TYPE "CW_DIG"
VERSION : 0.1
   STRUCT
      AUTO_CMD { ExternalWritable := 'False'} : Bool;   // Auto command
      FORCE : Bool;   // Force command
      SPARE { ExternalAccessible := 'False'; ExternalVisible := 'False'; ExternalWritable := 'False'} : Bool;
      ENABLE { S7_SetPoint := 'True'} : Bool;   // Master enable
      SPARE4 { ExternalAccessible := 'False'; ExternalVisible := 'False'; ExternalWritable := 'False'} : Bool;
      INPUT { ExternalWritable := 'False'} : Bool;   // Input Status
      SPARE6 { ExternalAccessible := 'False'; ExternalVisible := 'False'; ExternalWritable := 'False'} : Bool;
      SPARE7 { ExternalAccessible := 'False'; ExternalVisible := 'False'; ExternalWritable := 'False'} : Bool;
      SPARE8 { ExternalAccessible := 'False'; ExternalVisible := 'False'; ExternalWritable := 'False'} : Bool;
      SPARE9 { ExternalAccessible := 'False'; ExternalVisible := 'False'; ExternalWritable := 'False'} : Bool;
      SPARE10 { ExternalAccessible := 'False'; ExternalVisible := 'False'; ExternalWritable := 'False'} : Bool;
      SPARE11 { ExternalAccessible := 'False'; ExternalVisible := 'False'; ExternalWritable := 'False'} : Bool;
      SPARE12 { ExternalAccessible := 'False'; ExternalVisible := 'False'; ExternalWritable := 'False'} : Bool;
      EXIST { S7_SetPoint := 'True'} : Bool;   // Exist
      OUT_ACT { ExternalWritable := 'False'} : Bool;   // Output activation
      SPARE15 { ExternalAccessible := 'False'; ExternalVisible := 'False'; ExternalWritable := 'False'} : Bool;
   END_STRUCT;

END_TYPE

TYPE "CW_MTR"
VERSION : 0.1
   STRUCT
      START_REQ { ExternalWritable := 'False'} : Bool;   // Start request
      FORCE : Bool;   // Force command
      RST_REQ : Bool;   // Reset request
      ENABLE { S7_SetPoint := 'True'} : Bool;   // Master enable
      FB_RDY { ExternalWritable := 'False'} : Bool;   // Feedback Ready/Trip
      FB_RUN { ExternalWritable := 'False'} : Bool;   // Feedback Run
      FB_RDY_EN { S7_SetPoint := 'True'} : Bool;   // Enable Ready/Trip Feedback
      FB_RUN_EN { S7_SetPoint := 'True'} : Bool;   // Enable Run Feedback
      SPARE9 { ExternalAccessible := 'False'; ExternalVisible := 'False'; ExternalWritable := 'False'} : Bool;
      NO_ERR { ExternalWritable := 'False'} : Bool;   // No error
      SRV_RST : Bool;   // Reset service interval
      SRV_IND { ExternalWritable := 'False'} : Bool;   // Service interval elapsed
      SPARE1 { ExternalAccessible := 'False'; ExternalVisible := 'False'; ExternalWritable := 'False'} : Bool;
      EXIST { S7_SetPoint := 'True'} : Bool;   // Exist
      OUT_ACT { ExternalWritable := 'False'} : Bool;   // Output activation
      SPARE2 { ExternalAccessible := 'False'; ExternalVisible := 'False'; ExternalWritable := 'False'} : Bool;
   END_STRUCT;

END_TYPE

TYPE "CW_AN"
VERSION : 0.1
   STRUCT
      SPARE0 { ExternalAccessible := 'False'; ExternalVisible := 'False'; ExternalWritable := 'False'} : Bool;
      FORCE : Bool;   // Force output
      SP_CHANGE : Bool;   // Setpoint change trigger
      ENABLE { S7_SetPoint := 'True'} : Bool;   // 1=Master enable
      SPARE4 { ExternalAccessible := 'False'; ExternalVisible := 'False'; ExternalWritable := 'False'} : Bool;
      OPEN { ExternalWritable := 'False'} : Bool;   // PLC request > 0.1
      SPARE6 { ExternalAccessible := 'False'; ExternalVisible := 'False'; ExternalWritable := 'False'} : Bool;
      SPARE7 { ExternalAccessible := 'False'; ExternalVisible := 'False'; ExternalWritable := 'False'} : Bool;
      SPARE8 { ExternalAccessible := 'False'; ExternalVisible := 'False'; ExternalWritable := 'False'} : Bool;
      NO_ERR { ExternalWritable := 'False'} : Bool;   // 1=No error
      PAR_CHANGE : Bool;   // Parameter change trigger
      SPARE11 { ExternalAccessible := 'False'; ExternalVisible := 'False'; ExternalWritable := 'False'} : Bool;
      NO { S7_SetPoint := 'True'} : Bool;   // 0=NC, 1=NO
      EXIST { S7_SetPoint := 'True'} : Bool;   // 1=Exist
      SPARE14 { ExternalAccessible := 'False'; ExternalVisible := 'False'; ExternalWritable := 'False'} : Bool;
      SPARE15 { ExternalAccessible := 'False'; ExternalVisible := 'False'; ExternalWritable := 'False'} : Bool;
   END_STRUCT;

END_TYPE

TYPE "CW_VLV"
VERSION : 0.1
   STRUCT
      AUTO_CMD { ExternalWritable := 'False'} : Bool;   // Auto command
      FORCE : Bool;   // Force command
      SPARE2 { ExternalAccessible := 'False'; ExternalVisible := 'False'; ExternalWritable := 'False'} : Bool;   // Setpoint change indication
      ENABLE { S7_SetPoint := 'True'} : Bool;   // Master enable
      FB_CLS { ExternalWritable := 'False'} : Bool;   // Feedback Close
      FB_OPN { ExternalWritable := 'False'} : Bool;   // Feedback Open
      FB_CLS_EN { S7_SetPoint := 'True'} : Bool;   // Enable Close Feedback
      FB_OPN_EN { S7_SetPoint := 'True'} : Bool;   // Enable Open Feedback
      OPN_REQ { ExternalWritable := 'False'} : Bool;   // Open Request
      NO_ERR { ExternalWritable := 'False'} : Bool;   // No error
      SRV_RST : Bool;   // Reset service interval
      SRV_IND { ExternalWritable := 'False'} : Bool;   // Service interval elapsed
      NO { S7_SetPoint := 'True'} : Bool;   // NO/NC
      EXIST { S7_SetPoint := 'True'} : Bool;   // Valve exist
      OUT_ACT { ExternalWritable := 'False'} : Bool;   // Output activation
      VLV_W_FB { S7_SetPoint := 'True'} : Bool;   // Valve without position feedbacks
   END_STRUCT;

END_TYPE

TYPE "STAT MTR"
VERSION : 0.1
   STRUCT
      TAG { ExternalWritable := 'False'; S7_SetPoint := 'True'} : String[10];   // Tag label
      CW : "CW_MTR";   // Control/Status Word
      RUN_HRS { ExternalWritable := 'False'} : UInt;   // Runtime
      FB_RUN_ADD { S7_SetPoint := 'True'} : Int := 8;   // Input address - run feedback
      FB_RDY_ADD { S7_SetPoint := 'True'} : Int := 8;   // Input address - trip feedback
      OUT_ACT_ADD { S7_SetPoint := 'True'} : Int := 8;   // Output address - activation
   END_STRUCT;

END_TYPE

TYPE "STAT VLV"
VERSION : 0.1
   STRUCT
      TAG { ExternalWritable := 'False'; S7_SetPoint := 'True'} : String[10];   // Valve tag label
      CW { S7_SetPoint := 'False'} : "CW_VLV";   // Control/Status word
      SERV_CNTR { ExternalWritable := 'False'; S7_SetPoint := 'True'} : Int;
      FB_OPN_ADD { S7_SetPoint := 'True'} : Int := 8;   // Input address - open position feedback
      FB_CLS_ADD { S7_SetPoint := 'True'} : Int := 8;   // Input address - closed position feedback
      ACT_OUT_ADD { S7_SetPoint := 'True'} : Int := 8;   // Output address - activation
   END_STRUCT;

END_TYPE

TYPE "STAT AO"
VERSION : 0.1
   STRUCT
      Tag { ExternalWritable := 'False'; S7_SetPoint := 'True'} : String[10];   // Tag label
      CW : "CW_AN";
      "Type" { ExternalAccessible := 'False'; ExternalVisible := 'False'; ExternalWritable := 'False'; S7_SetPoint := 'True'} : SInt;   // 0=V/mA, 1=Spare, 2=PN
      Address { S7_SetPoint := 'True'} : Int;   // Output Address
      Min { S7_SetPoint := 'True'} : Real;   // Scaled Min
      Max { S7_SetPoint := 'True'} : Real;   // Scaled Max
      CV : Real;   // Output value
      EU { ExternalWritable := 'False'; S7_SetPoint := 'True'} : Int;   // Eng Unit
   END_STRUCT;

END_TYPE

TYPE "STAT AI"
VERSION : 0.1
   STRUCT
      Tag { ExternalWritable := 'False'; S7_SetPoint := 'True'} : String[10];   // Tag label
      CW : "CW_AN";   // Control Word
      "Type" { S7_SetPoint := 'True'} : SInt;   // 0 = V/mA; 1 = RTD; 2=PN
      Address { S7_SetPoint := 'True'} : Int;   // Input Address
      Min { S7_SetPoint := 'True'} : Real;   // Scale min
      Max { S7_SetPoint := 'True'} : Real;   // Scale max
      PV { ExternalWritable := 'False'} : Real;   // Process value
      EU { ExternalWritable := 'False'; S7_SetPoint := 'True'} : Int;   // Engineering Units
   END_STRUCT;

END_TYPE

TYPE "STAT DI"
VERSION : 0.1
   STRUCT
      Tag { ExternalWritable := 'False'; S7_SetPoint := 'True'} : String[10];   // Tag label
      CW : "CW_DIG";
      Address { S7_SetPoint := 'True'} : Int := 8;   // Input address
   END_STRUCT;

END_TYPE

TYPE "STAT DO"
VERSION : 0.1
   STRUCT
      Tag { ExternalWritable := 'False'; S7_SetPoint := 'True'} : String[10];   // Tag label
      CW : "CW_DIG";
      Address { S7_SetPoint := 'True'} : Int := 8;   // Output address
   END_STRUCT;

END_TYPE

TYPE "STAT VFD"
VERSION : 0.1
   STRUCT
      TAG { ExternalWritable := 'False'; S7_SetPoint := 'True'} : String[10];   // Tag label
      CW : "CW_MTR";   // Control/Status Word
      "TYPE" { S7_SetPoint := 'True'} : Int;   // 0=DOL, 1=Hardwired, 2=ABB PN,  3=DANFOSS PN
      RUN_HRS { ExternalWritable := 'False'} : UInt;   // Runtime
      FB_RUN_ADD { S7_SetPoint := 'True'} : Int := 8;   // Run feedback input address
      FB_RDY_ADD { S7_SetPoint := 'True'} : Int := 8;   // Trip feedback input address
      OUT_ACT_ADD { S7_SetPoint := 'True'} : Int := 8;   // Start output address
      OUT_RST_ADD { S7_SetPoint := 'True'} : Int := 8;   // Reset output address
   END_STRUCT;

END_TYPE

TYPE "EM - 210"
VERSION : 0.1
   STRUCT
      "AV210-1" { ExternalAccessible := 'False'; ExternalVisible := 'False'; ExternalWritable := 'False'} : "STAT VLV" := ('AV210-1', ((), (), (), (), (), (), TRUE, TRUE, (), (), (), (), (), TRUE, (), TRUE), (), 184, 185, 162);   // Recirculation on/off line
      "FCV210-1" { ExternalAccessible := 'False'; ExternalVisible := 'False'; ExternalWritable := 'False'} : "STAT AO" := ('FCV210-1', ((), (), (), (), (), (), (), (), (), (), (), (), (), (), (), ()), 0, 74, (), 100.0, (), 5);   // Recirculation control valve
   END_STRUCT;

END_TYPE

TYPE "EM - 375"
VERSION : 0.1
   STRUCT
      "AV37X-1" { ExternalAccessible := 'False'; ExternalVisible := 'False'; ExternalWritable := 'False'} : "STAT VLV" := ('AV375-1', ((), (), (), TRUE, (), (), (), (), (), (), (), (), (), TRUE, (), ()), (), 8, 8, 325);   // Op. water supply
      LS793 { ExternalAccessible := 'False'; ExternalVisible := 'False'; ExternalWritable := 'False'} : "STAT DI" := ('LS793', ((), (), (), (), (), (), (), (), (), (), (), (), (), True, (), ()), 167);   // Make-up water level
      "PIS375-1" { ExternalAccessible := 'False'; ExternalVisible := 'False'; ExternalWritable := 'False'} : "STAT DI" := ('PIS375-1', ((), (), (), TRUE, (), (), (), (), (), (), (), (), (), TRUE, (), ()), 165);   // Op. water pressure
      "PT37X-1" { ExternalAccessible := 'False'; ExternalVisible := 'False'; ExternalWritable := 'False'} : "STAT AI" := ('PT376-1', ((), (), (), (), (), (), (), (), (), (), (), (), (), True, (), ()), 0, 102, 0.0, 1000.0, (), ());   // Op. water pressure
   END_STRUCT;

END_TYPE

TYPE "EM - 506"
VERSION : 0.1
   STRUCT
      "AV543-1" { ExternalAccessible := 'False'; ExternalVisible := 'False'; ExternalWritable := 'False'} : "STAT VLV" := ('AV543-1', ((), (), (), (), (), (), TRUE, TRUE, (), (), (), (), TRUE, TRUE, (), TRUE), (), 220, 221, 180);   // Cyclone vent pipe
      IP506a { ExternalAccessible := 'False'; ExternalVisible := 'False'; ExternalWritable := 'False'} : "STAT AO" := ('IP506A', ((), (), (), (), (), (), (), (), (), (), (), (), (), True, (), ()), (), 68, (), 100.0, (), 5);   // Discharge pressure
      "PV376-1" { ExternalAccessible := 'False'; ExternalVisible := 'False'; ExternalWritable := 'False'} : "STAT VLV" := ('PV376-1', ((), (), (), (), (), (), (), (), (), (), (), (), (), TRUE, (), ()), (), 8, 8, 337);   // Op. water supply
      "PV376-2" { ExternalAccessible := 'False'; ExternalVisible := 'False'; ExternalWritable := 'False'} : "STAT VLV" := ('PV376-2', ((), (), (), (), (), (), (), (), (), (), (), (), (), TRUE, (), ()), (), 8, 8, 340);   // Op. water supply
      AVDCH { ExternalAccessible := 'False'; ExternalVisible := 'False'; ExternalWritable := 'False'} : "STAT VLV" := ('506c', ((), (), (), TRUE, (), (), (), (), (), (), (), (), (), TRUE, (), ()), (), (), (), 332);   // Large discharge
   END_STRUCT;

END_TYPE

TYPE "EM - P201"
VERSION : 0.1
   STRUCT
      "P201-1" { ExternalAccessible := 'False'; ExternalVisible := 'False'; ExternalWritable := 'False'} : "STAT VFD" := ('P201-1', ((), (), (), (), (), (), TRUE, TRUE, (), (), (), (), (), TRUE, (), ()), 1, (), 346, 347, 246, 247);   // Feed pump
      "P201-1_SPEED_REF" { ExternalAccessible := 'False'; ExternalVisible := 'False'; ExternalWritable := 'False'} : "STAT AO" := ((), ((), (), (), (), (), (), (), (), (), (), (), (), (), (), (), ()), (), 82, (), 100.0, (), 5);
      "TS201-1" { ExternalAccessible := 'False'; ExternalVisible := 'False'; ExternalWritable := 'False'} : "STAT DI" := ('TS201-1', ((), (), (), (), (), (), (), (), (), (), (), (), (), (), (), ()), ());   // PTC for feed pump motor
   END_STRUCT;

END_TYPE

TYPE "EM - 208"
VERSION : 0.1
   STRUCT
      "AV208-1" { ExternalAccessible := 'False'; ExternalVisible := 'False'; ExternalWritable := 'False'} : "STAT VLV" := ('AV208-1', ((), (), (), (), (), (), TRUE, TRUE, (), (), (), (), (), (), (), TRUE), (), 182, 183, 161);   // Blending line on/off valve
      "FCV208-1" { ExternalAccessible := 'False'; ExternalVisible := 'False'; ExternalWritable := 'False'} : "STAT AO" := ('FCV208-1', ((), (), (), (), (), (), (), (), (), (), (), (), (), (), (), ()), 0, 72, (), 100.0, (), 5);   // Blending flow control valve
      "FIT208-1" { ExternalAccessible := 'False'; ExternalVisible := 'False'; ExternalWritable := 'False'} : "STAT AI" := ('FIT208-1', ((), (), (), (), (), (), (), (), (), (), (), (), (), (), (), ()), (), (), (), (), (), ());   // Blending flow meter
      "P208-1" { ExternalAccessible := 'False'; ExternalVisible := 'False'; ExternalWritable := 'False'} : "STAT MTR" := ('P208-1', ((), (), (), (), (), (), TRUE, TRUE, (), (), (), (), (), TRUE, (), ()), (), 350, 351, 250);   // Blending pump
      "QT220-2" { ExternalAccessible := 'False'; ExternalVisible := 'False'; ExternalWritable := 'False'} : "STAT AI" := ('QT220-2', ((), (), (), (), (), (), (), (), (), (), (), (), (), (), (), ()), 0, 86, 0.0, 1000.0, (), ());   // Blending turbidity
      "QT220-2_OK" { ExternalAccessible := 'False'; ExternalVisible := 'False'; ExternalWritable := 'False'} : "STAT DI" := ((), ((), (), (), (), (), (), (), (), (), (), (), (), (), (), (), ()), 173);   // Turbicity sensor status
   END_STRUCT;

END_TYPE

TYPE "EM - 300"
VERSION : 0.1
   STRUCT
      "AV301-1" { ExternalAccessible := 'False'; ExternalVisible := 'False'; ExternalWritable := 'False'} : "STAT VLV" := ('AV301-1', ((), (), (), TRUE, (), (), TRUE, TRUE, (), (), (), (), (), TRUE, (), TRUE), (), 200, 201, 170);   // Flush water supply
      "AV302a-1" { ExternalAccessible := 'False'; ExternalVisible := 'False'; ExternalWritable := 'False'} : "STAT VLV" := ('AV302a-1', ((), (), (), (), (), (), (), (), (), (), (), (), (), (), (), ()), (), (), (), 164);   // Flush above bowl
      "AV302-1" { ExternalAccessible := 'False'; ExternalVisible := 'False'; ExternalWritable := 'False'} : "STAT VLV" := ('AV302-1', ((), (), (), (), (), (), (), (), (), (), (), (), (), TRUE, (), ()), (), 8, 8, 320);   // Flush bowl upper
      "AV303-1" { ExternalAccessible := 'False'; ExternalVisible := 'False'; ExternalWritable := 'False'} : "STAT VLV" := ('AV303-1', ((), (), (), (), (), (), (), (), (), (), (), (), (), TRUE, (), ()), (), 8, 8, 321);   // Flush bowl lower
      "AV304-1" { ExternalAccessible := 'False'; ExternalVisible := 'False'; ExternalWritable := 'False'} : "STAT VLV" := ('AV304-1', ((), (), (), (), (), (), (), (), (), (), (), (), (), TRUE, (), ()), (), 8, 8, 322);   // Flush sediment outlet
      "AV305-1" { ExternalAccessible := 'False'; ExternalVisible := 'False'; ExternalWritable := 'False'} : "STAT VLV" := ('AV305-1', ((), (), (), (), (), (), (), (), (), (), (), (), (), TRUE, (), ()), (), 8, 8, 323);   // Flush cyclone
      "AV306-1" { ExternalAccessible := 'False'; ExternalVisible := 'False'; ExternalWritable := 'False'} : "STAT VLV" := ('AV306-1', ((), (), (), (), (), (), (), (), (), (), (), (), (), TRUE, (), ()), (), 8, 8, 324);   // Flush cyclone vent pipe
      "AV320-1" { ExternalAccessible := 'False'; ExternalVisible := 'False'; ExternalWritable := 'False'} : "STAT VLV" := ('AV320-1', ((), (), (), (), (), (), TRUE, TRUE, (), (), (), (), (), TRUE, (), TRUE), (), 202, 203, 171);   // CIP flush supply
      "AV635-1" { ExternalAccessible := 'False'; ExternalVisible := 'False'; ExternalWritable := 'False'} : "STAT VLV" := ('AV635-1', ((), (), (), (), (), (), (), (), (), (), (), (), (), TRUE, (), ()), (), 8, 8, 330);   // Flush outlet mechanical seals
      "PS301-1" { ExternalAccessible := 'False'; ExternalVisible := 'False'; ExternalWritable := 'False'} : "STAT DI" := ('PS301-1', ((), (), (), (), (), (), (), (), (), (), (), (), (), True, (), ()), 164);   // Water supply pressure
   END_STRUCT;

END_TYPE

TYPE "EM - PRU2"
VERSION : 0.1
   STRUCT
      "AV460b-1" { ExternalAccessible := 'False'; ExternalVisible := 'False'; ExternalWritable := 'False'} : "STAT VLV" := ('AV460b-1', ((), (), (), (), (), (), (), (), (), (), (), (), TRUE, TRUE, (), ()), (), (), (), 162);   // PRU tank drain
      "AV660b-1" { ExternalAccessible := 'False'; ExternalVisible := 'False'; ExternalWritable := 'False'} : "STAT VLV" := ('AV660b-1', ((), (), (), (), (), (), (), (), (), (), (), (), (), TRUE, (), ()), (), (), (), 192);   // Sealing liquid SRU pump
      "GS220-1" { ExternalAccessible := 'False'; ExternalVisible := 'False'; ExternalWritable := 'False'} : "STAT DI" := ('GS220-1', ((), (), (), (), (), (), (), (), (), (), (), (), (), (), (), ()), 186);   // PRU tank cover switch
      "FS661b-1" { ExternalAccessible := 'False'; ExternalVisible := 'False'; ExternalWritable := 'False'} : "STAT DI" := ((), ((), (), (), (), (), (), (), (), (), (), (), (), (), (), (), ()), 172);   // PRU sealing l
      "P220-1" { ExternalAccessible := 'False'; ExternalVisible := 'False'; ExternalWritable := 'False'} : "STAT VFD" := ('P220-1', ((), (), (), (), (), (), TRUE, TRUE, (), (), (), (), (), TRUE, (), ()), 2, (), (), (), 540, ());   // PRU pump
   END_STRUCT;

END_TYPE

TYPE "EM - 463"
VERSION : 0.1
   STRUCT
      "AV305-2" { ExternalAccessible := 'False'; ExternalVisible := 'False'; ExternalWritable := 'False'} : "STAT VLV" := ('AV305-2', ((), (), (), (), (), (), (), (), (), (), (), (), (), TRUE, (), ()), (), 8, 8, 345);   // Tank flush - CIP
      "AV463-1" { ExternalAccessible := 'False'; ExternalVisible := 'False'; ExternalWritable := 'False'} : "STAT VLV" := ('AV463-1', ((), (), (), (), (), (), TRUE, TRUE, (), (), (), (), TRUE, TRUE, (), TRUE), (), 224, 225, 182);   // Inlet valve
      "AV463-2" { ExternalAccessible := 'False'; ExternalVisible := 'False'; ExternalWritable := 'False'} : "STAT VLV" := ('AV463-2', ((), (), (), (), (), (), TRUE, TRUE, (), (), (), (), (), TRUE, (), TRUE), (), 226, 227, 183);   // Overflow outlet valve
      "AV470-1" { ExternalAccessible := 'False'; ExternalVisible := 'False'; ExternalWritable := 'False'} : "STAT VLV" := ('AV470-1', ((), (), (), (), (), (), (), (), (), (), (), (), TRUE, TRUE, (), ()), (), 8, 8, 342);   // Pressure relief valve
      "AV660-1" { ExternalAccessible := 'False'; ExternalVisible := 'False'; ExternalWritable := 'False'} : "STAT VLV" := ('AV660-1', ((), (), (), (), (), (), (), (), (), (), (), (), (), TRUE, (), ()), (), 8, 8, 341);   // Vacuum pump sealing water
      "AV660-2" { ExternalAccessible := 'False'; ExternalVisible := 'False'; ExternalWritable := 'False'} : "STAT VLV" := ('AV660-2', ((), (), (), (), (), (), (), (), (), (), (), (), (), TRUE, (), ()), (), 8, 8, 346);   // Tank flush - water
      "LT463-1" { ExternalAccessible := 'False'; ExternalVisible := 'False'; ExternalWritable := 'False'} : "STAT AI" := ('LT463-1', ((), (), (), (), (), (), (), (), (), (), (), (), (), (), (), ()), (), 82, (), 100.0, (), ());   // Tank level
      "PIT463-1" { ExternalAccessible := 'False'; ExternalVisible := 'False'; ExternalWritable := 'False'} : "STAT AI" := ('PIT463-1', ((), (), (), (), (), (), (), (), (), (), (), (), (), (), (), ()), (), 84, -100.0, 1000.0, (), ());   // eMotion pressure
      "P463-1" { ExternalAccessible := 'False'; ExternalVisible := 'False'; ExternalWritable := 'False'} : "STAT MTR" := ('P463-1', ((), (), (), (), (), (), TRUE, TRUE, (), (), (), (), (), TRUE, (), ()), (), 344, 345, 245);   // Vacuum pump
   END_STRUCT;

END_TYPE

TYPE "EM - 551"
VERSION : 0.1
   STRUCT
      "FIT551-1" { ExternalAccessible := 'False'; ExternalVisible := 'False'; ExternalWritable := 'False'} : "STAT AI" := ('FIT551-1', ((), (), (), (), (), (), (), (), (), (), (), (), (), (), (), ()), (), 66, (), 70700.0, (), ());   // ProCarb CO2 flowmeter
      "FCV551-1" { ExternalAccessible := 'False'; ExternalVisible := 'False'; ExternalWritable := 'False'} : "STAT AO" := ('FCV551-1', ((), (), (), (), (), (), (), (), (), (), (), (), (), (), (), ()), (), 66, (), 100.0, (), 5);   // ProCarb CO2 flow control valve
   END_STRUCT;

END_TYPE

TYPE "EM - PRU1"
VERSION : 0.1
   STRUCT
      "AV461b-1" { ExternalAccessible := 'False'; ExternalVisible := 'False'; ExternalWritable := 'False'} : "STAT VLV" := ('AV461b-1', ((), (), (), (), (), (), (), (), (), (), (), (), TRUE, TRUE, (), ()), (), (), (), 163);   // PRU tank drain
      "AV660a-1" { ExternalAccessible := 'False'; ExternalVisible := 'False'; ExternalWritable := 'False'} : "STAT VLV" := ('AV660a-1', ((), (), (), (), (), (), (), (), (), (), (), (), (), TRUE, (), ()), (), (), (), 191);   // Sealing liquid SRU pump
      "GS221-1" { ExternalAccessible := 'False'; ExternalVisible := 'False'; ExternalWritable := 'False'} : "STAT DI" := ('GS221-1', ((), (), (), (), (), (), (), (), (), (), (), (), (), (), (), ()), 187);   // PRU cover switch
      "FS661a-1" { ExternalAccessible := 'False'; ExternalVisible := 'False'; ExternalWritable := 'False'} : "STAT DI" := ((), ((), (), (), (), (), (), (), (), (), (), (), (), (), (), (), ()), 171);
      "P221-1" { ExternalAccessible := 'False'; ExternalVisible := 'False'; ExternalWritable := 'False'} : "STAT VFD" := ('P221-1', ((), (), (), (), (), (), TRUE, TRUE, (), (), (), (), (), TRUE, (), ()), 2, (), (), (), 532, ());   // PRU pump
   END_STRUCT;

END_TYPE

TYPE "EM - 222"
VERSION : 0.1
   STRUCT
      "AV222-1" { ExternalAccessible := 'False'; ExternalVisible := 'False'; ExternalWritable := 'False'} : "STAT VLV" := ('AV222-1', ((), (), (), (), (), (), TRUE, TRUE, (), (), (), (), (), TRUE, (), TRUE), (), 194, 195, 166);   // Soilds outlet change-over valve
      "LS222-1" { ExternalAccessible := 'False'; ExternalVisible := 'False'; ExternalWritable := 'False'} : "STAT DI" := ('LS222-1', ((), (), (), TRUE, (), (), (), (), (), (), (), (), (), True, (), ()), 326);   // Level in cyclone high-high
      "LS222-2" { ExternalAccessible := 'False'; ExternalVisible := 'False'; ExternalWritable := 'False'} : "STAT DI" := ('LS222-2', ((), (), (), (), (), (), (), (), (), (), (), (), (), (), (), ()), 327);   // Level in cylone high
      "LS222-3" { ExternalAccessible := 'False'; ExternalVisible := 'False'; ExternalWritable := 'False'} : "STAT DI" := ('LS222-3', ((), (), (), (), (), (), (), (), (), (), (), (), (), (), (), ()), 330);   // Level in cyclone low
      "P222-1" { ExternalAccessible := 'False'; ExternalVisible := 'False'; ExternalWritable := 'False'} : "STAT MTR" := ('P222-1', ((), (), (), TRUE, (), (), TRUE, TRUE, (), (), (), (), (), True, (), ()), (), 334, 335, 242);   // Solids pump
      "PIT222-1" { ExternalAccessible := 'False'; ExternalVisible := 'False'; ExternalWritable := 'False'} : "STAT AI" := ('PIT222-1', ((), (), (), (), (), (), (), (), (), (), (), (), (), (), (), ()), (), 78, (), 1000.0, (), ());   // Solids pressure
      "TS222-1" { ExternalAccessible := 'False'; ExternalVisible := 'False'; ExternalWritable := 'False'} : "STAT DI" := ('TS222-1', ((), (), (), TRUE, (), (), (), (), (), (), (), (), (), TRUE, (), ()), 324);   // Solids pump dry-run potection
      "TT222-1" { ExternalAccessible := 'False'; ExternalVisible := 'False'; ExternalWritable := 'False'} : "STAT AI" := ('TT222-1', ((), (), (), (), (), (), (), (), (), (), (), (), (), (), (), ()), 1, 134, 0.0, 200.0, (), ());   // Solids pump stator temperature
   END_STRUCT;

END_TYPE

TYPE "EM - BC-COMM"
VERSION : 0.1
   STRUCT
      BCI0 { ExternalAccessible := 'False'; ExternalVisible := 'False'; ExternalWritable := 'False'; S7_SetPoint := 'True'} : Int := 173;   // BC I/O CMD
      BCI1 { ExternalAccessible := 'False'; ExternalVisible := 'False'; ExternalWritable := 'False'; S7_SetPoint := 'True'} : Int := 174;   // BC I/O CMD
      BCI2 { ExternalAccessible := 'False'; ExternalVisible := 'False'; ExternalWritable := 'False'; S7_SetPoint := 'True'} : Int := 175;   // BC I/O CMD
      BCI3 { ExternalAccessible := 'False'; ExternalVisible := 'False'; ExternalWritable := 'False'; S7_SetPoint := 'True'} : Int := 176;   // BC I/O CMD
      BCO0 { ExternalAccessible := 'False'; ExternalVisible := 'False'; ExternalWritable := 'False'; S7_SetPoint := 'True'} : Int := 185;   // BC I/O STATUS
      BCO1 { ExternalAccessible := 'False'; ExternalVisible := 'False'; ExternalWritable := 'False'; S7_SetPoint := 'True'} : Int := 186;   // BC I/O STATUS
      BCO2 { ExternalAccessible := 'False'; ExternalVisible := 'False'; ExternalWritable := 'False'; S7_SetPoint := 'True'} : Int := 187;   // BC I/O STATUS
      BCO3 { ExternalAccessible := 'False'; ExternalVisible := 'False'; ExternalWritable := 'False'; S7_SetPoint := 'True'} : Int := 190;   // BC I/O STATUS
      ALARM { ExternalAccessible := 'False'; ExternalVisible := 'False'; ExternalWritable := 'False'; S7_SetPoint := 'True'} : Int := 197;   // BC I/O STATUS
   END_STRUCT;

END_TYPE

TYPE "EM - RCB"
VERSION : 0.1
   STRUCT
      "RCB_IN_Dch 1" { ExternalAccessible := 'False'; ExternalVisible := 'False'; ExternalWritable := 'False'; S7_SetPoint := 'True'} : Int := 200;   // RCB CMD
      "RCB_IN_Dch 2" { ExternalAccessible := 'False'; ExternalVisible := 'False'; ExternalWritable := 'False'; S7_SetPoint := 'True'} : Int := 201;   // RCB CMD
      RCB_IN_ZoomIn { ExternalAccessible := 'False'; ExternalVisible := 'False'; ExternalWritable := 'False'; S7_SetPoint := 'True'} : Int := 202;   // RCB CMD
      RCB_IN_Prod { ExternalAccessible := 'False'; ExternalVisible := 'False'; ExternalWritable := 'False'; S7_SetPoint := 'True'} : Int := 203;   // RCB CMD
      RCB_IN_WaterTest { ExternalAccessible := 'False'; ExternalVisible := 'False'; ExternalWritable := 'False'; S7_SetPoint := 'True'} : Int := 204;   // RCB CMD
      RCB_IN_CipWater { ExternalAccessible := 'False'; ExternalVisible := 'False'; ExternalWritable := 'False'; S7_SetPoint := 'True'} : Int := 205;   // RCB CMD
      RCB_IN_ZoomOut { ExternalAccessible := 'False'; ExternalVisible := 'False'; ExternalWritable := 'False'; S7_SetPoint := 'True'} : Int := 206;   // RCB CMD
      RCB_IN_Start { ExternalAccessible := 'False'; ExternalVisible := 'False'; ExternalWritable := 'False'; S7_SetPoint := 'True'} : Int := 207;   // RCB CMD
      RCB_IN_Stop { ExternalAccessible := 'False'; ExternalVisible := 'False'; ExternalWritable := 'False'; S7_SetPoint := 'True'} : Int := 210;   // RCB CMD
      ExtInterlockStart { ExternalAccessible := 'False'; ExternalVisible := 'False'; ExternalWritable := 'False'; S7_SetPoint := 'True'} : Int := 160;   // INTERLOCKS
      ExtInterlockProd { ExternalAccessible := 'False'; ExternalVisible := 'False'; ExternalWritable := 'False'; S7_SetPoint := 'True'} : Int := 161;   // INTERLOCKS
      ExtInterlockCIP { ExternalAccessible := 'False'; ExternalVisible := 'False'; ExternalWritable := 'False'; S7_SetPoint := 'True'} : Int := 162;   // INTERLOCKS
      "RCB_OUT_Dch 1" { ExternalAccessible := 'False'; ExternalVisible := 'False'; ExternalWritable := 'False'; S7_SetPoint := 'True'} : Int := 160;   // RCB STATUS
      "RCB_OUT_Dch 2" { ExternalAccessible := 'False'; ExternalVisible := 'False'; ExternalWritable := 'False'; S7_SetPoint := 'True'} : Int := 161;   // RCB STATUS
      RCB_OUT_ZoomIn { ExternalAccessible := 'False'; ExternalVisible := 'False'; ExternalWritable := 'False'; S7_SetPoint := 'True'} : Int := 162;   // RCB STATUS
      RCB_OUT_Prod { ExternalAccessible := 'False'; ExternalVisible := 'False'; ExternalWritable := 'False'; S7_SetPoint := 'True'} : Int := 163;   // RCB STATUS
      RCB_OUT_WaterTest { ExternalAccessible := 'False'; ExternalVisible := 'False'; ExternalWritable := 'False'; S7_SetPoint := 'True'} : Int := 164;   // RCB STATUS
      RCB_OUT_CipWater { ExternalAccessible := 'False'; ExternalVisible := 'False'; ExternalWritable := 'False'; S7_SetPoint := 'True'} : Int := 165;   // RCB STATUS
      RCB_OUT_ZoomOut { ExternalAccessible := 'False'; ExternalVisible := 'False'; ExternalWritable := 'False'; S7_SetPoint := 'True'} : Int := 166;   // RCB STATUS
      RCB_OUT_Start { ExternalAccessible := 'False'; ExternalVisible := 'False'; ExternalWritable := 'False'; S7_SetPoint := 'True'} : Int := 167;   // RCB STATUS
      RCB_OUT_Stop { ExternalAccessible := 'False'; ExternalVisible := 'False'; ExternalWritable := 'False'; S7_SetPoint := 'True'} : Int := 170;   // RCB STATUS
   END_STRUCT;

END_TYPE

TYPE "EM - 430"
VERSION : 0.1
   STRUCT
      "AV400-1" { ExternalAccessible := 'False'; ExternalVisible := 'False'; ExternalWritable := 'False'} : "STAT VLV" := ('AV400-1', ((), (), (), (), (), (), (), (), (), (), (), (), (), TRUE, (), ()), (), 8, 8, 8);   // Cooling liquid supply
      "AV430-1" { ExternalAccessible := 'False'; ExternalVisible := 'False'; ExternalWritable := 'False'} : "STAT VLV" := ('AV430-1', ((), (), (), (), (), (), (), (), (), (), (), (), (), TRUE, (), ()), (), 8, 8, 343);   // Glycol supply
      "FCV430-1" { ExternalAccessible := 'False'; ExternalVisible := 'False'; ExternalWritable := 'False'} : "STAT AO" := ('FCV430-1', ((), (), (), (), (), (), (), (), (), (), (), (), (), (), (), ()), (), 76, (), 100.0, (), 5);   // Glycol flow control valve
      "LT406-1" { ExternalAccessible := 'False'; ExternalVisible := 'False'; ExternalWritable := 'False'} : "STAT AI" := ('LT406-1', ((), (), (), (), (), (), (), (), (), (), (), (), (), (), (), ()), (), (), (), 100.0, (), ());   // Cooling liquid level
      "P406-1" { ExternalAccessible := 'False'; ExternalVisible := 'False'; ExternalWritable := 'False'} : "STAT MTR" := ('P406-1', ((), (), (), (), (), (), TRUE, TRUE, (), (), (), (), (), TRUE, (), ()), (), 342, 343, 244);   // Cooling liquid pump
      "TT406-1" { ExternalAccessible := 'False'; ExternalVisible := 'False'; ExternalWritable := 'False'} : "STAT AI" := ('TT406-1', ((), (), (), (), (), (), (), (), (), (), (), (), (), (), (), ()), (), 86, (), 200.0, (), ());   // Cooling liquid temperature
   END_STRUCT;

END_TYPE

TYPE "EM - 212"
VERSION : 0.1
   STRUCT
      "AV212-1" { ExternalAccessible := 'False'; ExternalVisible := 'False'; ExternalWritable := 'False'} : "STAT VLV" := ('AV212-1', ((), (), (), (), (), (), TRUE, TRUE, (), (), (), (), TRUE, TRUE, (), TRUE), (), 186, 187, 163);   // By-pass valve
   END_STRUCT;

END_TYPE

TYPE "EM - 206"
VERSION : 0.1
   STRUCT
      "AV206-1" : "STAT VLV" := ('AV206-1', ((), (), (), (), (), (), (), (), (), (), (), (), (), True, (), ()), (), 8, 8, 161);   // Brine/Centrate on/off valve
      "PIT206-1" : "STAT AI" := ('PIT206-1', ((), (), (), (), (), (), (), (), (), (), (), (), (), True, (), ()), 0, 86, 0.0, 1000.0, (), ());   // Brine/Centrate pressure
   END_STRUCT;

END_TYPE

TYPE "EM - 22X"
VERSION : 0.1
   STRUCT
      "AV220-1" { ExternalAccessible := 'False'; ExternalVisible := 'False'; ExternalWritable := 'False'} : "STAT VLV" := ('AV220-1', ((), (), (), (), (), (), TRUE, TRUE, (), (), (), (), (), TRUE, (), TRUE), (), 190, 191, 164);   // LP outlet valve
      "AV460-1" { ExternalAccessible := 'False'; ExternalVisible := 'False'; ExternalWritable := 'False'} : "STAT VLV" := ('AV460-1', ((), (), (), (), (), (), TRUE, TRUE, (), (), (), (), TRUE, TRUE, (), TRUE), (), 210, 211, 174);   // LP outlet to drain valve
      "SV220-1" { ExternalAccessible := 'False'; ExternalVisible := 'False'; ExternalWritable := 'False'} : "STAT VLV" := ('SV220-1', ((), (), (), (), (), (), (), (), (), (), (), (), (), (), (), ()), (), (), (), 333);   // Back pressure air supply
      "FIT22X-1" { ExternalAccessible := 'False'; ExternalVisible := 'False'; ExternalWritable := 'False'} : "STAT AI" := ('FIT220-1', ((), (), (), True, (), (), (), (), (), (), (), (), (), (), (), ()), (), (), (), (), (), ());   // LP outlet flowmeter
      "PIT22X-1" { ExternalAccessible := 'False'; ExternalVisible := 'False'; ExternalWritable := 'False'} : "STAT AI" := ('PIT220-1', ((), (), (), True, (), (), (), (), (), (), (), (), (), True, (), ()), 0, 66, 0.0, 1000.0, (), ());   // LP outlet pressure
      "QT220-1" { ExternalAccessible := 'False'; ExternalVisible := 'False'; ExternalWritable := 'False'} : "STAT AI" := ('QT220-1', ((), (), (), (), (), (), (), (), (), (), (), (), (), True, (), ()), 0, 70, 0.0, 100.0, (), ());   // LP outlet turbidity
      "PCV22X-1" { ExternalAccessible := 'False'; ExternalVisible := 'False'; ExternalWritable := 'False'} : "STAT AO" := ('PCV220-1', ((), (), (), True, (), (), (), (), (), (), (), (), (), True, (), ()), 0, 66, (), 100.0, (), 5);   // LP outlet pressure control valve
      "QT220-1_OK" { ExternalAccessible := 'False'; ExternalVisible := 'False'; ExternalWritable := 'False'} : "STAT DI" := ('QT220-1 OK', ((), (), (), (), (), (), (), (), (), (), (), (), (), True, (), ()), 172);   // Turbidity sensor status
      "LA220-1" { ExternalAccessible := 'False'; ExternalVisible := 'False'; ExternalWritable := 'False'} : "STAT DO" := ('LA220-1', ((), (), (), (), (), (), (), (), (), (), (), (), (), True, (), ()), 192);   // LP outlet sight glass backlight
   END_STRUCT;

END_TYPE

TYPE "EM - 100"
VERSION : 0.1
   STRUCT
      "L-GREEN" { ExternalAccessible := 'False'; ExternalVisible := 'False'; ExternalWritable := 'False'} : "STAT DO" := ('L-GREEN', ((), (), (), (), (), (), (), (), (), (), (), (), (), True, (), ()), 193);   // Green light
      "L-YELLOW" { ExternalAccessible := 'False'; ExternalVisible := 'False'; ExternalWritable := 'False'} : "STAT DO" := ('L-YELLOW', ((), (), (), (), (), (), (), (), (), (), (), (), (), True, (), ()), 194);   // Yellow light
      "L-RED" { ExternalAccessible := 'False'; ExternalVisible := 'False'; ExternalWritable := 'False'} : "STAT DO" := ('L-RED', ((), (), (), TRUE, (), (), (), (), (), (), (), (), (), TRUE, (), ()), 195);   // Red light
      "L-BUZZ" { ExternalAccessible := 'False'; ExternalVisible := 'False'; ExternalWritable := 'False'} : "STAT DO" := ('L-BUZZ', ((), (), (), TRUE, (), (), (), (), (), (), (), (), (), TRUE, (), ()), 196);   // Buzzier
      EMS { ExternalAccessible := 'False'; ExternalVisible := 'False'; ExternalWritable := 'False'} : "STAT DI" := ('E-STOP', ((), (), (), TRUE, (), (), (), (), (), (), (), (), (), TRUE, (), ()), 320);   // E-stop
      UPS { ExternalAccessible := 'False'; ExternalVisible := 'False'; ExternalWritable := 'False'} : "STAT DI" := ('UPS', ((), (), (), TRUE, (), (), (), (), (), (), (), (), (), (), (), ()), 321);   // UPS battery
      EWON { ExternalAccessible := 'False'; ExternalVisible := 'False'; ExternalWritable := 'False'} : "STAT DI" := ('eWON', ((), (), (), (), (), (), (), (), (), (), (), (), (), (), (), ()), 177);   // eWON Talk2M status
      "CA VIB WARN" { ExternalAccessible := 'False'; ExternalVisible := 'False'; ExternalWritable := 'False'} : "STAT DI" := ('CA WARN', ((), (), (), (), (), (), (), (), (), (), (), (), (), (), (), ()), 360);   // Vibration pre-warning
      "CA VIB ALM" { ExternalAccessible := 'False'; ExternalVisible := 'False'; ExternalWritable := 'False'} : "STAT DI" := ('CA ALM', ((), (), (), (), (), (), (), (), (), (), (), (), (), (), (), ()), 361);   // Vibration alarm
      "CA ERROR" { ExternalAccessible := 'False'; ExternalVisible := 'False'; ExternalWritable := 'False'} : "STAT DI" := ('CA ERROR', ((), (), (), (), (), (), (), (), (), (), (), (), (), (), (), ()), 362);   // Error status
      "CA WD" { ExternalAccessible := 'False'; ExternalVisible := 'False'; ExternalWritable := 'False'} : "STAT DI" := ('CA WD', ((), (), (), (), (), (), (), (), (), (), (), (), (), (), (), ()), 363);   // Watchdog
      "PS502-1" { ExternalAccessible := 'False'; ExternalVisible := 'False'; ExternalWritable := 'False'} : "STAT DI" := ('PS502-1', ((), (), (), TRUE, (), (), (), (), (), (), (), (), (), TRUE, (), ()), 166);   // Instrument air supply
      "LT BUF" { ExternalAccessible := 'False'; ExternalVisible := 'False'; ExternalWritable := 'False'} : "STAT AI" := ('LT BUF', ((), (), (), TRUE, (), (), (), (), (), (), (), (), (), (), (), ()), (), 80, (), 100.0, (), 5);   // Buffer tank level
   END_STRUCT;

END_TYPE

TYPE "EM - 400"
VERSION : 0.1
   STRUCT
      "AV409-1" { ExternalAccessible := 'False'; ExternalVisible := 'False'; ExternalWritable := 'False'} : "STAT VLV" := ('AV409-1', ((), (), (), True, (), (), (), (), (), (), (), (), (), True, (), ()), (), 8, 8, 326);   // Cooling liquid supply
      "FCV409-1" { ExternalAccessible := 'False'; ExternalVisible := 'False'; ExternalWritable := 'False'} : "STAT AO" := ('FCV409-1', ((), (), (), (), (), (), (), (), (), (), (), (), (), True, (), ()), (), 78, (), 100.0, (), 5);   // Dynamic cooling flow control valve
      "FIS409-1" { ExternalAccessible := 'False'; ExternalVisible := 'False'; ExternalWritable := 'False'} : "STAT DI" := ('FIS409-1', ((), (), (), True, (), (), (), (), (), (), (), (), (), True, (), ()), 160);   // Cooling liquid flow
      "FIS412-1" { ExternalAccessible := 'False'; ExternalVisible := 'False'; ExternalWritable := 'False'} : "STAT DI" := ('FIS412-1', ((), (), (), (), (), (), (), (), (), (), (), (), (), True, (), ()), 366);   // Cooling liquid flow
      "FIT409-1" { ExternalAccessible := 'False'; ExternalVisible := 'False'; ExternalWritable := 'False'} : "STAT AI" := ('FIT409-1', ((), (), (), (), (), (), (), (), (), (), (), (), (), True, (), ()), (), 92, 0.0, 240.0, (), ());   // Dynamic cooling flow
      "FIT412-1" { ExternalAccessible := 'False'; ExternalVisible := 'False'; ExternalWritable := 'False'} : "STAT AI" := ('FIT412-1', ((), (), (), (), (), (), (), (), (), (), (), (), (), True, (), ()), 0, 100, 0.0, 1500.0, (), ());   // Cooling liquid flow
      "TT411-1" { ExternalAccessible := 'False'; ExternalVisible := 'False'; ExternalWritable := 'False'} : "STAT AI" := ('TT411-1', ((), (), (), (), (), (), (), (), (), (), (), (), (), True, (), ()), 1, 136, 0.0, 200.0, (), ());   // Cooling liquid temperature
      "TT41X-1" { ExternalAccessible := 'False'; ExternalVisible := 'False'; ExternalWritable := 'False'} : "STAT AI" := ('TT410-1', ((), (), (), (), (), (), (), (), (), (), (), (), (), True, (), ()), 1, 142, (), 200.0, (), ());   // Cooling liquid temperature
   END_STRUCT;

END_TYPE

TYPE "EM - 420"
VERSION : 0.1
   STRUCT
      FS421a { ExternalAccessible := 'False'; ExternalVisible := 'False'; ExternalWritable := 'False'} : "STAT DI" := ('FS421a', ((), (), (), (), (), (), (), (), (), (), (), (), (), True, (), ()), 367);   // Oil flow top bearing
      FS421b { ExternalAccessible := 'False'; ExternalVisible := 'False'; ExternalWritable := 'False'} : "STAT DI" := ('FS421b', ((), (), (), (), (), (), (), (), (), (), (), (), (), True, (), ()), 370);   // Oil flow bottom bearing
      LS422a { ExternalAccessible := 'False'; ExternalVisible := 'False'; ExternalWritable := 'False'} : "STAT DI" := ('LS422a', ((), (), (), (), (), (), (), (), (), (), (), (), (), True, (), ()), 371);   // High oil level
      "LS42X(b)" { ExternalAccessible := 'False'; ExternalVisible := 'False'; ExternalWritable := 'False'} : "STAT DI" := ('LS422b', ((), (), (), (), (), (), (), (), (), (), (), (), (), True, (), ()), 372);   // Low oil level
      "LS422-1" { ExternalAccessible := 'False'; ExternalVisible := 'False'; ExternalWritable := 'False'} : "STAT DI" := ('LS422-1', ((), (), (), (), (), (), (), (), (), (), (), (), (), True, (), ()), 373);   // Water in the oil
      "P403-1" { ExternalAccessible := 'False'; ExternalVisible := 'False'; ExternalWritable := 'False'} : "STAT MTR" := ('P403-1', ((), (), (), (), (), (), True, True, (), (), (), (), (), True, (), ()), (), 340, 341, 243);   // Oil recirc pump
      "P421-1" { ExternalAccessible := 'False'; ExternalVisible := 'False'; ExternalWritable := 'False'} : "STAT MTR" := ('P421-1', ((), (), (), (), (), (), (), (), (), (), (), (), (), True, (), ()), (), (), (), 336);   // Lubricating pump
      "PS421-1" { ExternalAccessible := 'False'; ExternalVisible := 'False'; ExternalWritable := 'False'} : "STAT DI" := ('PS421-1', ((), (), (), (), (), (), (), (), (), (), (), (), (), True, (), ()), 374);   // Air pressure lubrication
      "PV421-1" { ExternalAccessible := 'False'; ExternalVisible := 'False'; ExternalWritable := 'False'} : "STAT VLV" := ('PV421-1', ((), (), (), (), (), (), (), (), (), (), (), (), (), True, (), ()), (), 8, 8, 335);   // Top bearing cooling
      "SV421-1" { ExternalAccessible := 'False'; ExternalVisible := 'False'; ExternalWritable := 'False'} : "STAT VLV" := ('SV421-1', ((), (), (), (), (), (), (), (), (), (), (), (), (), True, (), ()), (), (), (), 334);   // Air supply for lubricating system
   END_STRUCT;

END_TYPE

TYPE "EM - 508"
VERSION : 0.1
   STRUCT
      GS794 { ExternalAccessible := 'False'; ExternalVisible := 'False'; ExternalWritable := 'False'} : "STAT AI" := ('GS794', ((), (), (), (), (), (), (), (), (), (), (), (), (), True, (), ()), (), 64, (), 100.0, (), ());   // Centrizoom Position
      IP508b { ExternalAccessible := 'False'; ExternalVisible := 'False'; ExternalWritable := 'False'} : "STAT AO" := ('IP508B', ((), (), (), (), (), (), (), (), (), (), (), (), (), True, (), ()), (), 70, (), 100.0, (), ());   // Centrizoom Positioner
      "SV508b-1" { ExternalAccessible := 'False'; ExternalVisible := 'False'; ExternalWritable := 'False'} : "STAT VLV" := ('SV508b-1', ((), (), (), (), (), (), (), (), (), (), (), (), (), (), (), ()), (), (), (), 336);   // Centrizoom air supply
   END_STRUCT;

END_TYPE

TYPE "EM - 460"
VERSION : 0.1
   STRUCT
      "AV460d-1" { ExternalAccessible := 'False'; ExternalVisible := 'False'; ExternalWritable := 'False'} : "STAT VLV" := ('AV460d-1', ((), (), (), (), (), (), TRUE, TRUE, (), (), (), (), TRUE, TRUE, (), TRUE), (), 210, 211, 176);   // Liquid seal drain
   END_STRUCT;

END_TYPE

TYPE "EM - 600"
VERSION : 0.1
   STRUCT
      "AV615-1" { ExternalAccessible := 'False'; ExternalVisible := 'False'; ExternalWritable := 'False'} : "STAT VLV" := ('AV615-1', ((), (), (), (), (), (), (), (), (), (), (), (), TRUE, TRUE, (), ()), (), 8, 8, 327);   // Sealing water supply
      "AV63X/441-1" { ExternalAccessible := 'False'; ExternalVisible := 'False'; ExternalWritable := 'False'} : "STAT VLV" := ('AV630-1', ((), (), (), (), (), (), (), (), (), (), (), (), TRUE, TRUE, (), ()), (), (), (), ());   // Sealing water supply
      "FIS615-1" { ExternalAccessible := 'False'; ExternalVisible := 'False'; ExternalWritable := 'False'} : "STAT DI" := ('FIS615-1', ((), (), (), (), (), (), (), (), (), (), (), (), (), TRUE, (), ()), 161);   // Sealing water flow inlet seal
      "FIS630-1" { ExternalAccessible := 'False'; ExternalVisible := 'False'; ExternalWritable := 'False'} : "STAT DI" := ('FIS630-1', ((), (), (), (), (), (), (), (), (), (), (), (), (), True, (), ()), 163);   // Sealing water flow outlet seal
      "FIS635-1" { ExternalAccessible := 'False'; ExternalVisible := 'False'; ExternalWritable := 'False'} : "STAT DI" := ('FIS635-1', ((), (), (), (), (), (), (), (), (), (), (), (), (), TRUE, (), ()), 162);   // Sealing water flow outlet seal
   END_STRUCT;

END_TYPE

TYPE "EM - 701"
VERSION : 0.1
   STRUCT
      M701 { ExternalAccessible := 'False'; ExternalVisible := 'False'; ExternalWritable := 'False'} : "STAT VFD" := ('SC701', ((), (), (), TRUE, (), (), TRUE, TRUE, (), (), (), (), (), TRUE, (), ()), 1, (), 333, 332, 240, 241);   // Main motor VFD
      M701_SPEED_REF { ExternalAccessible := 'False'; ExternalVisible := 'False'; ExternalWritable := 'False'} : "STAT AO" := ((), ((), (), (), TRUE, (), (), (), (), (), (), (), (), (), TRUE, (), ()), (), 80, (), 100.0, (), 5);
      M701_AMPS { ExternalAccessible := 'False'; ExternalVisible := 'False'; ExternalWritable := 'False'} : "STAT AI" := ((), ((), (), (), TRUE, (), (), (), (), (), (), (), (), (), (), (), ()), (), 96, (), 150.0, (), 6);
   END_STRUCT;

END_TYPE

TYPE "EM - 22Y"
VERSION : 0.1
   STRUCT
      "AV221-1" { ExternalAccessible := 'False'; ExternalVisible := 'False'; ExternalWritable := 'False'} : "STAT VLV" := ('AV221-1', ((), (), (), (), (), (), TRUE, TRUE, (), (), (), (), (), TRUE, (), TRUE), (), 192, 193, 165);   // HP outlet valve
      "AV461-1" { ExternalAccessible := 'False'; ExternalVisible := 'False'; ExternalWritable := 'False'} : "STAT VLV" := ('AV461-1', ((), (), (), (), (), (), TRUE, TRUE, (), (), (), (), TRUE, TRUE, (), TRUE), (), 230, 231, 184);   // HP outlet to drain valve
      "FIT22Y-1" { ExternalAccessible := 'False'; ExternalVisible := 'False'; ExternalWritable := 'False'} : "STAT AI" := ('FIT221-1', ((), (), (), (), (), (), (), (), (), (), (), (), (), TRUE, (), ()), (), (), (), (), (), ());   // HP outlet flow meter
      "LA221-1" { ExternalAccessible := 'False'; ExternalVisible := 'False'; ExternalWritable := 'False'} : "STAT DO" := ('LA221-1', ((), (), (), (), (), (), (), (), (), (), (), (), (), TRUE, (), ()), 197);   // LP outlet sight glass backlight
      "PCV22Y-1" { ExternalAccessible := 'False'; ExternalVisible := 'False'; ExternalWritable := 'False'} : "STAT AO" := ('PCV221-1', ((), (), (), (), (), (), (), (), (), (), (), (), TRUE, TRUE, (), ()), 0, 70, (), 100.0, (), 5);   // HP outlet pressure control valve
      "PIT22Y-1" { ExternalAccessible := 'False'; ExternalVisible := 'False'; ExternalWritable := 'False'} : "STAT AI" := ('PIT221-1', ((), (), (), (), (), (), (), (), (), (), (), (), (), TRUE, (), ()), 0, 76, 0.0, 1000.0, (), ());   // HP outlet pressure
      "QT221-1" { ExternalAccessible := 'False'; ExternalVisible := 'False'; ExternalWritable := 'False'} : "STAT AI" := ('QT221-1', ((), (), (), (), (), (), (), (), (), (), (), (), (), (), (), ()), (), (), (), 100.0, (), 5);   // HP Outlet turbidity
   END_STRUCT;

END_TYPE

TYPE "EM - 730"
VERSION : 0.1
   STRUCT
      TS730 { ExternalAccessible := 'False'; ExternalVisible := 'False'; ExternalWritable := 'False'} : "STAT DI" := ('TS730', ((), (), (), (), (), (), (), (), (), (), (), (), (), True, (), ()), 325);   // Motor temperature PTC
      TT730a { ExternalAccessible := 'False'; ExternalVisible := 'False'; ExternalWritable := 'False'} : "STAT AI" := ('TT730a', ((), (), (), (), (), (), (), (), (), (), (), (), (), True, (), ()), 1, 128, (), 200.0, (), ());   // Temperature sensor in motor winding, Pt100
      TT730b { ExternalAccessible := 'False'; ExternalVisible := 'False'; ExternalWritable := 'False'} : "STAT AI" := ('TT730b', ((), (), (), (), (), (), (), (), (), (), (), (), (), True, (), ()), 1, 138, (), 200.0, (), ());   // Temperature sensor in motor winding (LD) or air space (eDrive), Pt100
      TT731a { ExternalAccessible := 'False'; ExternalVisible := 'False'; ExternalWritable := 'False'} : "STAT AI" := ('TT731', ((), (), (), (), (), (), (), (), (), (), (), (), (), True, (), ()), 1, 130, (), 200.0, (), ());   // Temperature sensor, neck bearing, Pt100
      TT731b { ExternalAccessible := 'False'; ExternalVisible := 'False'; ExternalWritable := 'False'} : "STAT AI" := ('TT731b', ((), (), (), (), (), (), (), (), (), (), (), (), (), (), (), ()), 1, 132, (), 200.0, (), ());   // Temperature sensor, neck bearing, Pt100
      TT733 { ExternalAccessible := 'False'; ExternalVisible := 'False'; ExternalWritable := 'False'} : "STAT AI" := ('TT733', ((), (), (), (), (), (), (), (), (), (), (), (), (), True, (), ()), 1, 132, (), 200.0, (), ());   // Gear oil temperature Pt100
      TT734 { ExternalAccessible := 'False'; ExternalVisible := 'False'; ExternalWritable := 'False'} : "STAT AI" := ('TT734', ((), (), (), (), (), (), (), (), (), (), (), (), (), True, (), ()), 1, 140, (), 200.0, (), ());   // Bottom bearing temperature Pt100
   END_STRUCT;

END_TYPE

TYPE "EM - 750"
VERSION : 0.1
   STRUCT
      YT75X { ExternalAccessible := 'False'; ExternalVisible := 'False'; ExternalWritable := 'False'} : "STAT AI" := ('YT750', ((), (), (), True, (), (), (), (), (), (), (), (), (), True, (), ()), (), 98, (), 25.0, (), 50);   // Vibration: Frame
   END_STRUCT;

END_TYPE

TYPE "EM - 340"
VERSION : 0.1
   STRUCT
      "AV340-1" { ExternalAccessible := 'False'; ExternalVisible := 'False'; ExternalWritable := 'False'} : "STAT VLV" := ('AV340-1', ((), (), (), TRUE, (), (), TRUE, TRUE, (), (), (), (), (), TRUE, (), TRUE), (), 204, 205, 172);   // Safety water supply
      "AV340-2" { ExternalAccessible := 'False'; ExternalVisible := 'False'; ExternalWritable := 'False'} : "STAT VLV" := ('AV340-2', ((), (), (), (), (), (), TRUE, TRUE, (), (), (), (), (), TRUE, (), TRUE), (), 206, 207, 173);   // Safety water supply
      "AV460-2" { ExternalAccessible := 'False'; ExternalVisible := 'False'; ExternalWritable := 'False'} : "STAT VLV" := ('AV460-2', ((), (), (), (), (), (), TRUE, TRUE, (), (), (), (), TRUE, TRUE, (), TRUE), (), 212, 213, 175);   // Safety water to drain
      "PIS340-1" { ExternalAccessible := 'False'; ExternalVisible := 'False'; ExternalWritable := 'False'} : "STAT DI" := ('PIS340-1', ((), (), (), (), (), (), (), (), (), (), (), (), (), TRUE, (), ()), 164);   // Safety water pressure
      "V340-1" { ExternalAccessible := 'False'; ExternalVisible := 'False'; ExternalWritable := 'False'} : "STAT DI" := ('V340-1', ((), (), (), (), (), (), (), (), (), (), (), (), (), (), (), ()), ());   // Safety water manual valve
   END_STRUCT;

END_TYPE

TYPE "EM - 201"
VERSION : 0.1
   STRUCT
      "AV201-1" { ExternalAccessible := 'False'; ExternalVisible := 'False'; ExternalWritable := 'False'} : "STAT VLV" := ('AV201-1', ((), (), (), TRUE, (), (), TRUE, TRUE, (), (), (), (), (), TRUE, (), TRUE), (), 180, 181, 160);   // Inlet on/off valve
      "AV460a-1" { ExternalAccessible := 'False'; ExternalVisible := 'False'; ExternalWritable := 'False'} : "STAT VLV" := ('AV460a-1', ((), (), (), (), (), (), (), (), (), (), (), (), (), True, (), ()), (), (), (), 172);   // Inlet to drain
      "FCV201-1" { ExternalAccessible := 'False'; ExternalVisible := 'False'; ExternalWritable := 'False'} : "STAT AO" := ('FCV201-1', ((), (), (), TRUE, (), (), (), (), (), (), (), (), FALSE, TRUE, (), ()), 0, 64, (), 100.0, (), 5);   // Inlet flow control valve
      "FIT201-1" { ExternalAccessible := 'False'; ExternalVisible := 'False'; ExternalWritable := 'False'} : "STAT AI" := ('FIT201-1', ((), (), (), TRUE, (), (), (), (), (), (), (), (), (), TRUE, (), ()), (), (), (), (), (), ());   // Inlet flow meter
      "LA201-1" { ExternalAccessible := 'False'; ExternalVisible := 'False'; ExternalWritable := 'False'} : "STAT DO" := ('LA201-1', ((), (), (), TRUE, (), (), (), (), (), (), (), (), (), TRUE, (), ()), 191);   // Inlet sight glass backlight
      "PIT201-1" { ExternalAccessible := 'False'; ExternalVisible := 'False'; ExternalWritable := 'False'} : "STAT AI" := ('PIT201-1', ((), (), (), TRUE, (), (), (), (), (), (), (), (), (), TRUE, (), ()), 0, 64, 0.0, 1000.0, (), ());   // Inlet pressure
      "QT201-1" { ExternalAccessible := 'False'; ExternalVisible := 'False'; ExternalWritable := 'False'} : "STAT AI" := ('QT201-1', ((), (), (), (), (), (), (), (), (), (), (), (), (), (), (), ()), 0, 68, 0.0, 100.0, (), ());   // Inlet turbidity
      "TT201-1" { ExternalAccessible := 'False'; ExternalVisible := 'False'; ExternalWritable := 'False'} : "STAT AI" := ('TT201-1', ((), (), (), (), (), (), (), (), (), (), (), (), (), (), (), ()), (), (), (), 200.0, (), ());   // Inlet temperature
      "QT201-1_OK" { ExternalAccessible := 'False'; ExternalVisible := 'False'; ExternalWritable := 'False'} : "STAT DI" := ('QT201-1 OK', ((), (), (), (), (), (), (), (), (), (), (), (), (), (), (), ()), 171);   // Turbidity sensor OK
   END_STRUCT;

END_TYPE

TYPE "EM - 740"
VERSION : 0.1
   STRUCT
      "P+F PS" { ExternalAccessible := 'False'; ExternalVisible := 'False'; ExternalWritable := 'False'} : "STAT DO" := ('P+F PS', ((), (), (), TRUE, (), (), (), (), (), (), (), (), (), TRUE, (), ()), 252);   // Speed converter: Power supply
      "P+F OS" { ExternalAccessible := 'False'; ExternalVisible := 'False'; ExternalWritable := 'False'} : "STAT DI" := ('P+F OS', ((), (), (), TRUE, (), (), (), (), (), (), (), (), (), TRUE, (), ()), 322);   // Speed converter: Overspeed
      "P+F ERROR" { ExternalAccessible := 'False'; ExternalVisible := 'False'; ExternalWritable := 'False'} : "STAT DI" := ('P+F ERROR', ((), (), (), TRUE, (), (), (), (), (), (), (), (), (), TRUE, (), ()), 323);   // Speed converter: Error
   END_STRUCT;

END_TYPE

TYPE "MachineConfig"
VERSION : 0.1
   STRUCT
      "Family" { S7_SetPoint := 'True'} : Int;   // 1-Brew, 2-Clara, 3-CR, 4-PurePuls, 5-KR, 6-Protein, 7-VOT, 8-Dairy
      TypeNo { S7_SetPoint := 'True'} : Int;   // HSS ID number
      Range { ExternalWritable := 'False'; S7_SetPoint := 'True'} : Int;   // 1-TumbaL, 2-PuneS
      SepType { ExternalWritable := 'False'; S7_SetPoint := 'True'} : Int;   // 1-Clarifier, 2-Purifier, 3-Concentrator
      Frame { ExternalWritable := 'False'; S7_SetPoint := 'True'} : Int;   // 1=18, 2=18e, 3=15, 4=13, 5=10, 6=07, 7=04, 8=LD
      DchSystem { ExternalWritable := 'False'; S7_SetPoint := 'True'} : Int;   // 1-Dosing ring, 2-OWMC, 3-OWMCe, 4-OWM II
      Spare_1 { ExternalWritable := 'False'; S7_SetPoint := 'True'} : Int;
      FeedPump { S7_SetPoint := 'True'} : Int;   // 0-Not compatible, 1-Compatible, 2-Installed
      Blending { S7_SetPoint := 'True'} : Int;   // 0-Not compatible, 1-Compatible, 2-Installed
      Recirculation { S7_SetPoint := 'True'} : Int;   // 0-Not compatible, 1-Compatible, 2-Installed
      CoolingRecirculation { S7_SetPoint := 'True'} : Int;   // 0-Not compatible, 1-Compatible, 2-Installed
      Spare_2 { S7_SetPoint := 'True'} : Int;   // 0-Not compatible, 1-Compatible, 2-Installed
      eMotion { S7_SetPoint := 'True'} : Int;   // 0-Not compatible, 1-Compatible, 2-Installed
      InlineCarbonation { S7_SetPoint := 'True'} : Int;   // 0-Not compatible, 1-Compatible, 2-Installed
      ConditionAlert { S7_SetPoint := 'True'} : Int;   // 0-Not compatible, 1-Compatible, 2-Installed
      "PRU-1" { S7_SetPoint := 'True'} : Int;   // 0-Not compatible, 1-Compatible, 2-Installed
      "PRU-2" { S7_SetPoint := 'True'} : Int;   // 0-Not compatible, 1-Compatible, 2-Installed
      eWON { S7_SetPoint := 'True'} : Int;   // 0-Not compatible, 1-Compatible, 2-Installed
      ALBufferTank { S7_SetPoint := 'True'} : Int;   // 0-Not compatible, 1-Compatible, 2-Installed
      RCB { S7_SetPoint := 'True'} : Int;   // 0-Not compatible, 1-Compatible, 2-Installed
      Spare_3 { S7_SetPoint := 'True'} : Int;
   END_STRUCT;

END_TYPE

TYPE "STAT Dch"
VERSION : 0.1
   STRUCT
      "EM - 222" { ExternalAccessible := 'False'; ExternalVisible := 'False'; ExternalWritable := 'False'} : "EM - 222";   // SRU
      "EM - 300" { ExternalAccessible := 'False'; ExternalVisible := 'False'; ExternalWritable := 'False'} : "EM - 300";   // Flushing
      "EM - 375" { ExternalAccessible := 'False'; ExternalVisible := 'False'; ExternalWritable := 'False'} : "EM - 375";   // Op.water
      "EM - 506" { ExternalAccessible := 'False'; ExternalVisible := 'False'; ExternalWritable := 'False'} : "EM - 506";   // Discharge system
   END_STRUCT;

END_TYPE

TYPE "STAT Sep"
VERSION : 0.1
   STRUCT
      "EM - 100" { ExternalAccessible := 'False'; ExternalVisible := 'False'; ExternalWritable := 'False'} : "EM - 100";   // Utilities
      "EM - 400" { ExternalAccessible := 'False'; ExternalVisible := 'False'; ExternalWritable := 'False'} : "EM - 400";   // Cooling liquid
      "EM - 420" { ExternalAccessible := 'False'; ExternalVisible := 'False'; ExternalWritable := 'False'} : "EM - 420";   // Lubrication
      "EM - 460" { ExternalAccessible := 'False'; ExternalVisible := 'False'; ExternalWritable := 'False'} : "EM - 460";   // Liquid seal
      "EM - 600" { ExternalAccessible := 'False'; ExternalVisible := 'False'; ExternalWritable := 'False'} : "EM - 600";   // Sealing liquids
      "EM - 701" { ExternalAccessible := 'False'; ExternalVisible := 'False'; ExternalWritable := 'False'} : "EM - 701";   // Main drive
      "EM - 730" { ExternalAccessible := 'False'; ExternalVisible := 'False'; ExternalWritable := 'False'} : "EM - 730";   // Temperature supervision
      "EM - 740" { ExternalAccessible := 'False'; ExternalVisible := 'False'; ExternalWritable := 'False'} : "EM - 740";   // Speed supervision
      "EM - 750" { ExternalAccessible := 'False'; ExternalVisible := 'False'; ExternalWritable := 'False'} : "EM - 750";   // Vibration supervision
      "EM - 508" { ExternalAccessible := 'False'; ExternalVisible := 'False'; ExternalWritable := 'False'} : "EM - 508";
   END_STRUCT;

END_TYPE

TYPE "STAT Options"
VERSION : 0.1
   STRUCT
      "EM - P201" { ExternalAccessible := 'False'; ExternalVisible := 'False'; ExternalWritable := 'False'} : "EM - P201";   // Feed pump
      "EM - 208" { ExternalAccessible := 'False'; ExternalVisible := 'False'; ExternalWritable := 'False'} : "EM - 208";   // Blending
      "EM - 210" { ExternalAccessible := 'False'; ExternalVisible := 'False'; ExternalWritable := 'False'} : "EM - 210";   // Recirculation
      "EM - 430" { ExternalAccessible := 'False'; ExternalVisible := 'False'; ExternalWritable := 'False'} : "EM - 430";   // Cooling recirculation
      "EM - 463" { ExternalAccessible := 'False'; ExternalVisible := 'False'; ExternalWritable := 'False'} : "EM - 463";   // eMotion
      "EM - 551" { ExternalAccessible := 'False'; ExternalVisible := 'False'; ExternalWritable := 'False'} : "EM - 551";   // ProCarb
      "EM - PRU1" { ExternalAccessible := 'False'; ExternalVisible := 'False'; ExternalWritable := 'False'} : "EM - PRU1";   // PRU1
      "EM - PRU2" { ExternalAccessible := 'False'; ExternalVisible := 'False'; ExternalWritable := 'False'} : "EM - PRU2";   // PRU2
   END_STRUCT;

END_TYPE

TYPE "STAT Process"
VERSION : 0.1
   STRUCT
      "EM - 201" { ExternalAccessible := 'False'; ExternalVisible := 'False'; ExternalWritable := 'False'} : "EM - 201";   // Product inlet
      "EM - 206" { ExternalAccessible := 'False'; ExternalVisible := 'False'; ExternalWritable := 'False'} : "EM - 206";   // Brine/Centrate inlet
      "EM - 212" { ExternalAccessible := 'False'; ExternalVisible := 'False'; ExternalWritable := 'False'} : "EM - 212";   // Bypass
      "EM - 22X" { ExternalAccessible := 'False'; ExternalVisible := 'False'; ExternalWritable := 'False'} : "EM - 22X";   // LP outlet
      "EM - 22Y" { ExternalAccessible := 'False'; ExternalVisible := 'False'; ExternalWritable := 'False'} : "EM - 22Y";   // HP outlet
      "EM - 340" { ExternalAccessible := 'False'; ExternalVisible := 'False'; ExternalWritable := 'False'} : "EM - 340";   // Safety water
   END_STRUCT;

END_TYPE

TYPE "STAT Comm"
VERSION : 0.1
   STRUCT
      "EM - BC-COMM" { ExternalAccessible := 'False'; ExternalVisible := 'False'; ExternalWritable := 'False'} : "EM - BC-COMM";
      "EM - RCB" { ExternalAccessible := 'False'; ExternalVisible := 'False'; ExternalWritable := 'False'} : "EM - RCB";
   END_STRUCT;

END_TYPE

TYPE "STAT SYSTEM"
VERSION : 0.1
   STRUCT
      Machine : "MachineConfig";
      "Unit Sep" { ExternalAccessible := 'False'; ExternalVisible := 'False'; ExternalWritable := 'False'} : "STAT Sep";
      "Unit Process" { ExternalAccessible := 'False'; ExternalVisible := 'False'; ExternalWritable := 'False'} : "STAT Process";
      "Unit Dch" { ExternalAccessible := 'False'; ExternalVisible := 'False'; ExternalWritable := 'False'} : "STAT Dch";
      Options { ExternalAccessible := 'False'; ExternalVisible := 'False'; ExternalWritable := 'False'} : "STAT Options";
      Communications { ExternalAccessible := 'False'; ExternalVisible := 'False'; ExternalWritable := 'False'} : "STAT Comm";
   END_STRUCT;

END_TYPE

DATA_BLOCK "SysConfig_Lib_KR"
TITLE = System configuration library - KR
{ DB_Accessible_From_OPC_UA := 'FALSE' ;
 S7_Optimized_Access := 'TRUE' }
AUTHOR : DBV
FAMILY : FactorySettings
VERSION : 0.1
UNLINKED
NON_RETAIN
   VAR
      MachineConfig { ExternalAccessible := 'False'; ExternalVisible := 'False'; ExternalWritable := 'False'; S7_SetPoint := 'False'} : Array[0..5] of "STAT SYSTEM";
   END_VAR


BEGIN
   MachineConfig[0].Machine."Family" := 5;
   MachineConfig[0].Machine.TypeNo := 60;
   MachineConfig[0].Machine.Range := 2;
   MachineConfig[0].Machine.SepType := 1;
   MachineConfig[0].Machine.Frame := 1;
   MachineConfig[0].Machine.DchSystem := 2;
   MachineConfig[0].Machine.FeedPump := 1;
   MachineConfig[0].Machine.eWON := 1;
   MachineConfig[0]."Unit Sep"."EM - 100"."L-GREEN".CW.ENABLE := True;
   MachineConfig[0]."Unit Sep"."EM - 100"."L-GREEN".CW.EXIST := True;
   MachineConfig[0]."Unit Sep"."EM - 100"."L-YELLOW".Tag := 'L-BLUE';
   MachineConfig[0]."Unit Sep"."EM - 100"."L-RED".CW.ENABLE := True;
   MachineConfig[0]."Unit Sep"."EM - 100"."L-RED".CW.EXIST := True;
   MachineConfig[0]."Unit Sep"."EM - 100"."L-BUZZ".CW.ENABLE := True;
   MachineConfig[0]."Unit Sep"."EM - 100"."L-BUZZ".CW.EXIST := True;
   MachineConfig[0]."Unit Sep"."EM - 100".EMS.CW.ENABLE := True;
   MachineConfig[0]."Unit Sep"."EM - 100".EMS.CW.EXIST := True;
   MachineConfig[0]."Unit Sep"."EM - 100".EMS.Address := 180;
   MachineConfig[0]."Unit Sep"."EM - 100".UPS.CW.ENABLE := True;
   MachineConfig[0]."Unit Sep"."EM - 100".UPS.CW.EXIST := True;
   MachineConfig[0]."Unit Sep"."EM - 100".UPS.Address := 181;
   MachineConfig[0]."Unit Sep"."EM - 100".EWON.CW.ENABLE := True;
   MachineConfig[0]."Unit Sep"."EM - 100"."PS502-1".CW.ENABLE := True;
   MachineConfig[0]."Unit Sep"."EM - 100"."PS502-1".CW.EXIST := True;
   MachineConfig[0]."Unit Sep"."EM - 100"."LT BUF".CW.ENABLE := True;
   MachineConfig[0]."Unit Sep"."EM - 400"."AV409-1".CW.ENABLE := True;
   MachineConfig[0]."Unit Sep"."EM - 400"."AV409-1".CW.EXIST := True;
   MachineConfig[0]."Unit Sep"."EM - 400"."AV409-1".ACT_OUT_ADD := 170;
   MachineConfig[0]."Unit Sep"."EM - 400"."FCV409-1".CW.ENABLE := True;
   MachineConfig[0]."Unit Sep"."EM - 400"."FCV409-1".CW.EXIST := True;
   MachineConfig[0]."Unit Sep"."EM - 400"."FIS409-1".CW.ENABLE := False;
   MachineConfig[0]."Unit Sep"."EM - 400"."FIT409-1".CW.ENABLE := True;
   MachineConfig[0]."Unit Sep"."EM - 400"."FIT409-1".CW.EXIST := True;
   MachineConfig[0]."Unit Sep"."EM - 400"."TT41X-1".CW.ENABLE := True;
   MachineConfig[0]."Unit Sep"."EM - 400"."TT41X-1".CW.EXIST := True;
   MachineConfig[0]."Unit Sep"."EM - 400"."TT41X-1"."Type" := 0;
   MachineConfig[0]."Unit Sep"."EM - 400"."TT41X-1".Address := 86;
   MachineConfig[0]."Unit Sep"."EM - 400"."TT41X-1".Min := -50.0;
   MachineConfig[0]."Unit Sep"."EM - 400"."TT41X-1".Max := 150.0;
   MachineConfig[0]."Unit Sep"."EM - 600"."AV63X/441-1".TAG := 'AV441-1';
   MachineConfig[0]."Unit Sep"."EM - 600"."AV63X/441-1".CW.ENABLE := True;
   MachineConfig[0]."Unit Sep"."EM - 600"."AV63X/441-1".CW.EXIST := True;
   MachineConfig[0]."Unit Sep"."EM - 600"."AV63X/441-1".ACT_OUT_ADD := 174;
   MachineConfig[0]."Unit Sep"."EM - 701".M701.CW.ENABLE := True;
   MachineConfig[0]."Unit Sep"."EM - 701".M701.CW.FB_RDY_EN := True;
   MachineConfig[0]."Unit Sep"."EM - 701".M701.CW.FB_RUN_EN := True;
   MachineConfig[0]."Unit Sep"."EM - 701".M701.CW.EXIST := True;
   MachineConfig[0]."Unit Sep"."EM - 701".M701."TYPE" := 2;
   MachineConfig[0]."Unit Sep"."EM - 701".M701.FB_RUN_ADD := 8;
   MachineConfig[0]."Unit Sep"."EM - 701".M701.FB_RDY_ADD := 8;
   MachineConfig[0]."Unit Sep"."EM - 701".M701.OUT_ACT_ADD := 512;
   MachineConfig[0]."Unit Sep"."EM - 701".M701.OUT_RST_ADD := 8;
   MachineConfig[0]."Unit Sep"."EM - 701".M701_SPEED_REF.Address := 72;
   MachineConfig[0]."Unit Sep"."EM - 730".TS730.CW.ENABLE := True;
   MachineConfig[0]."Unit Sep"."EM - 730".TS730.CW.EXIST := True;
   MachineConfig[0]."Unit Sep"."EM - 730".TS730.Address := 184;
   MachineConfig[0]."Unit Sep"."EM - 740"."P+F PS".CW.ENABLE := True;
   MachineConfig[0]."Unit Sep"."EM - 740"."P+F PS".CW.EXIST := True;
   MachineConfig[0]."Unit Sep"."EM - 740"."P+F PS".Address := 180;
   MachineConfig[0]."Unit Sep"."EM - 740"."P+F OS".CW.ENABLE := True;
   MachineConfig[0]."Unit Sep"."EM - 740"."P+F OS".CW.EXIST := True;
   MachineConfig[0]."Unit Sep"."EM - 740"."P+F OS".Address := 182;
   MachineConfig[0]."Unit Sep"."EM - 740"."P+F ERROR".CW.ENABLE := True;
   MachineConfig[0]."Unit Sep"."EM - 740"."P+F ERROR".CW.EXIST := True;
   MachineConfig[0]."Unit Sep"."EM - 740"."P+F ERROR".Address := 183;
   MachineConfig[0]."Unit Sep"."EM - 750".YT75X.CW.ENABLE := True;
   MachineConfig[0]."Unit Sep"."EM - 750".YT75X.CW.EXIST := True;
   MachineConfig[0]."Unit Sep"."EM - 750".YT75X.Address := 78;
   MachineConfig[0]."Unit Process"."EM - 201"."AV201-1".CW.ENABLE := True;
   MachineConfig[0]."Unit Process"."EM - 201"."AV201-1".CW.FB_CLS_EN := False;
   MachineConfig[0]."Unit Process"."EM - 201"."AV201-1".CW.FB_OPN_EN := False;
   MachineConfig[0]."Unit Process"."EM - 201"."AV201-1".CW.EXIST := True;
   MachineConfig[0]."Unit Process"."EM - 201"."AV201-1".CW.VLV_W_FB := False;
   MachineConfig[0]."Unit Process"."EM - 201"."AV201-1".FB_OPN_ADD := 8;
   MachineConfig[0]."Unit Process"."EM - 201"."AV201-1".FB_CLS_ADD := 8;
   MachineConfig[0]."Unit Process"."EM - 201"."FCV201-1".CW.ENABLE := True;
   MachineConfig[0]."Unit Process"."EM - 201"."FCV201-1".CW.EXIST := True;
   MachineConfig[0]."Unit Process"."EM - 201"."FIT201-1".CW.ENABLE := True;
   MachineConfig[0]."Unit Process"."EM - 201"."FIT201-1".CW.EXIST := True;
   MachineConfig[0]."Unit Process"."EM - 201"."FIT201-1".Address := 88;
   MachineConfig[0]."Unit Process"."EM - 201"."FIT201-1".Max := 40000.0;
   MachineConfig[0]."Unit Process"."EM - 201"."LA201-1".CW.ENABLE := False;
   MachineConfig[0]."Unit Process"."EM - 201"."PIT201-1".CW.ENABLE := False;
   MachineConfig[0]."Unit Process"."EM - 22X"."AV220-1".CW.ENABLE := True;
   MachineConfig[0]."Unit Process"."EM - 22X"."AV220-1".CW.FB_CLS_EN := False;
   MachineConfig[0]."Unit Process"."EM - 22X"."AV220-1".CW.FB_OPN_EN := False;
   MachineConfig[0]."Unit Process"."EM - 22X"."AV220-1".CW.EXIST := True;
   MachineConfig[0]."Unit Process"."EM - 22X"."AV220-1".CW.VLV_W_FB := False;
   MachineConfig[0]."Unit Process"."EM - 22X"."AV220-1".FB_OPN_ADD := 8;
   MachineConfig[0]."Unit Process"."EM - 22X"."AV220-1".FB_CLS_ADD := 8;
   MachineConfig[0]."Unit Process"."EM - 22X"."AV220-1".ACT_OUT_ADD := 162;
   MachineConfig[0]."Unit Process"."EM - 22X"."AV460-1".CW.ENABLE := True;
   MachineConfig[0]."Unit Process"."EM - 22X"."AV460-1".CW.FB_CLS_EN := False;
   MachineConfig[0]."Unit Process"."EM - 22X"."AV460-1".CW.FB_OPN_EN := False;
   MachineConfig[0]."Unit Process"."EM - 22X"."AV460-1".CW.EXIST := True;
   MachineConfig[0]."Unit Process"."EM - 22X"."AV460-1".CW.VLV_W_FB := False;
   MachineConfig[0]."Unit Process"."EM - 22X"."AV460-1".FB_OPN_ADD := 8;
   MachineConfig[0]."Unit Process"."EM - 22X"."AV460-1".FB_CLS_ADD := 8;
   MachineConfig[0]."Unit Process"."EM - 22X"."AV460-1".ACT_OUT_ADD := 171;
   MachineConfig[0]."Unit Process"."EM - 22X"."FIT22X-1".CW.ENABLE := False;
   MachineConfig[0]."Unit Process"."EM - 22X"."PIT22X-1".CW.ENABLE := False;
   MachineConfig[0]."Unit Process"."EM - 22X"."PCV22X-1".CW.ENABLE := False;
   MachineConfig[0]."Unit Process"."EM - 340"."AV340-1".CW.ENABLE := True;
   MachineConfig[0]."Unit Process"."EM - 340"."AV340-1".CW.FB_CLS_EN := False;
   MachineConfig[0]."Unit Process"."EM - 340"."AV340-1".CW.FB_OPN_EN := False;
   MachineConfig[0]."Unit Process"."EM - 340"."AV340-1".CW.EXIST := True;
   MachineConfig[0]."Unit Process"."EM - 340"."AV340-1".CW.VLV_W_FB := False;
   MachineConfig[0]."Unit Process"."EM - 340"."AV340-1".FB_OPN_ADD := 8;
   MachineConfig[0]."Unit Process"."EM - 340"."AV340-1".FB_CLS_ADD := 8;
   MachineConfig[0]."Unit Process"."EM - 340"."AV340-1".ACT_OUT_ADD := 165;
   MachineConfig[0]."Unit Dch"."EM - 222"."LS222-1".CW.ENABLE := False;
   MachineConfig[0]."Unit Dch"."EM - 222"."LS222-1".Address := 185;
   MachineConfig[0]."Unit Dch"."EM - 222"."P222-1".CW.ENABLE := False;
   MachineConfig[0]."Unit Dch"."EM - 222"."P222-1".CW.FB_RDY_EN := True;
   MachineConfig[0]."Unit Dch"."EM - 222"."P222-1".CW.FB_RUN_EN := True;
   MachineConfig[0]."Unit Dch"."EM - 222"."P222-1".CW.EXIST := False;
   MachineConfig[0]."Unit Dch"."EM - 222"."P222-1".FB_RUN_ADD := 194;
   MachineConfig[0]."Unit Dch"."EM - 222"."P222-1".FB_RDY_ADD := 195;
   MachineConfig[0]."Unit Dch"."EM - 222"."P222-1".OUT_ACT_ADD := 182;
   MachineConfig[0]."Unit Dch"."EM - 300"."AV301-1".CW.ENABLE := True;
   MachineConfig[0]."Unit Dch"."EM - 300"."AV301-1".CW.FB_CLS_EN := False;
   MachineConfig[0]."Unit Dch"."EM - 300"."AV301-1".CW.FB_OPN_EN := False;
   MachineConfig[0]."Unit Dch"."EM - 300"."AV301-1".CW.EXIST := True;
   MachineConfig[0]."Unit Dch"."EM - 300"."AV301-1".CW.VLV_W_FB := False;
   MachineConfig[0]."Unit Dch"."EM - 300"."AV301-1".FB_OPN_ADD := 8;
   MachineConfig[0]."Unit Dch"."EM - 300"."AV301-1".FB_CLS_ADD := 8;
   MachineConfig[0]."Unit Dch"."EM - 300"."AV301-1".ACT_OUT_ADD := 163;
   MachineConfig[0]."Unit Dch"."EM - 300"."AV320-1".CW.ENABLE := True;
   MachineConfig[0]."Unit Dch"."EM - 300"."AV320-1".CW.FB_CLS_EN := False;
   MachineConfig[0]."Unit Dch"."EM - 300"."AV320-1".CW.FB_OPN_EN := False;
   MachineConfig[0]."Unit Dch"."EM - 300"."AV320-1".CW.EXIST := True;
   MachineConfig[0]."Unit Dch"."EM - 300"."AV320-1".CW.VLV_W_FB := False;
   MachineConfig[0]."Unit Dch"."EM - 300"."AV320-1".FB_OPN_ADD := 8;
   MachineConfig[0]."Unit Dch"."EM - 300"."AV320-1".FB_CLS_ADD := 8;
   MachineConfig[0]."Unit Dch"."EM - 300"."AV320-1".ACT_OUT_ADD := 164;
   MachineConfig[0]."Unit Dch"."EM - 375"."AV37X-1".CW.ENABLE := True;
   MachineConfig[0]."Unit Dch"."EM - 375"."AV37X-1".CW.EXIST := True;
   MachineConfig[0]."Unit Dch"."EM - 375"."AV37X-1".ACT_OUT_ADD := 166;
   MachineConfig[0]."Unit Dch"."EM - 375"."PIS375-1".CW.ENABLE := False;
   MachineConfig[0]."Unit Dch"."EM - 375"."PT37X-1".CW.ENABLE := True;
   MachineConfig[0]."Unit Dch"."EM - 375"."PT37X-1".CW.EXIST := True;
   MachineConfig[0]."Unit Dch"."EM - 375"."PT37X-1".Address := 76;
   MachineConfig[0]."Unit Dch"."EM - 375"."PT37X-1".Max := 600.0;
   MachineConfig[0]."Unit Dch"."EM - 506".IP506a.CW.ENABLE := True;
   MachineConfig[0]."Unit Dch"."EM - 506".IP506a.CW.EXIST := True;
   MachineConfig[0]."Unit Dch"."EM - 506".AVDCH.TAG := '506b';
   MachineConfig[0]."Unit Dch"."EM - 506".AVDCH.CW.ENABLE := True;
   MachineConfig[0]."Unit Dch"."EM - 506".AVDCH.CW.EXIST := True;
   MachineConfig[0]."Unit Dch"."EM - 506".AVDCH.ACT_OUT_ADD := 167;
   MachineConfig[0].Options."EM - P201"."P201-1".FB_RUN_ADD := 196;
   MachineConfig[0].Options."EM - P201"."P201-1".FB_RDY_ADD := 197;
   MachineConfig[0].Options."EM - P201"."P201-1".OUT_ACT_ADD := 183;
   MachineConfig[0].Options."EM - P201"."P201-1".OUT_RST_ADD := 184;
   MachineConfig[0].Options."EM - P201"."P201-1_SPEED_REF".Address := 70;
   MachineConfig[1].Machine."Family" := 5;
   MachineConfig[1].Machine.TypeNo := 61;
   MachineConfig[1].Machine.Range := 2;
   MachineConfig[1].Machine.SepType := 1;
   MachineConfig[1].Machine.Frame := 1;
   MachineConfig[1].Machine.DchSystem := 2;
   MachineConfig[1].Machine.Spare_1 := 3;
   MachineConfig[1].Machine.FeedPump := 1;
   MachineConfig[1].Machine.Spare_2 := 1;
   MachineConfig[1].Machine.ConditionAlert := 1;
   MachineConfig[1].Machine.eWON := 1;
   MachineConfig[1]."Unit Sep"."EM - 400"."AV409-1".CW.ENABLE := true;
   MachineConfig[1]."Unit Sep"."EM - 400"."FCV409-1".CW.ENABLE := True;
   MachineConfig[1]."Unit Sep"."EM - 400"."FIT409-1".CW.ENABLE := True;
   MachineConfig[1]."Unit Sep"."EM - 400"."TT41X-1".CW.ENABLE := True;
   MachineConfig[1]."Unit Sep"."EM - 600"."FIS615-1".CW.ENABLE := False;
   MachineConfig[1]."Unit Sep"."EM - 730".TS730.CW.ENABLE := true;
   MachineConfig[1]."Unit Sep"."EM - 730".TT731a.CW.ENABLE := True;
   MachineConfig[1]."Unit Sep"."EM - 750".YT75X.CW.ENABLE := TRUE;
   MachineConfig[1]."Unit Process"."EM - 201"."AV201-1".CW.ENABLE := True;
   MachineConfig[1]."Unit Process"."EM - 201"."FIT201-1"."Type" := 2;
   MachineConfig[1]."Unit Process"."EM - 201"."FIT201-1".Address := 256;
   MachineConfig[1]."Unit Process"."EM - 201"."FIT201-1".Max := 50000.0;
   MachineConfig[1]."Unit Process"."EM - 212"."AV212-1".CW.ENABLE := True;
   MachineConfig[1]."Unit Process"."EM - 22X"."AV220-1".CW.ENABLE := True;
   MachineConfig[1]."Unit Process"."EM - 22X"."AV460-1".CW.ENABLE := True;
   MachineConfig[1]."Unit Process"."EM - 22X"."PCV22X-1".CW.ENABLE := True;
   MachineConfig[1]."Unit Process"."EM - 22X"."PCV22X-1".CW.EXIST := True;
   MachineConfig[1]."Unit Process"."EM - 22X"."PCV22X-1".Address := 66;
   MachineConfig[1]."Unit Process"."EM - 22X"."LA220-1".CW.ENABLE := True;
   MachineConfig[1]."Unit Process"."EM - 340"."AV340-1".CW.ENABLE := True;
   MachineConfig[1]."Unit Process"."EM - 340"."AV340-2".CW.ENABLE := True;
   MachineConfig[1]."Unit Process"."EM - 340"."AV460-2".CW.ENABLE := true;
   MachineConfig[1]."Unit Dch"."EM - 222"."P222-1".CW.EXIST := False;
   MachineConfig[1]."Unit Dch"."EM - 222"."TS222-1".CW.ENABLE := true;
   MachineConfig[1]."Unit Dch"."EM - 300"."AV301-1".CW.ENABLE := True;
   MachineConfig[1]."Unit Dch"."EM - 300"."AV303-1".CW.ENABLE := True;
   MachineConfig[1]."Unit Dch"."EM - 300"."AV304-1".CW.ENABLE := True;
   MachineConfig[1]."Unit Dch"."EM - 300"."AV305-1".CW.ENABLE := True;
   MachineConfig[1]."Unit Dch"."EM - 300"."AV320-1".CW.ENABLE := True;
   MachineConfig[1]."Unit Dch"."EM - 375"."AV37X-1".CW.ENABLE := True;
   MachineConfig[1]."Unit Dch"."EM - 506".IP506a.CW.ENABLE := True;
   MachineConfig[1]."Unit Dch"."EM - 506".AVDCH.CW.ENABLE := True;
   MachineConfig[5]."Unit Process"."EM - 22X"."FIT22X-1".CW.ENABLE := True;
   MachineConfig[5]."Unit Process"."EM - 22X"."FIT22X-1".CW.EXIST := false;
   MachineConfig[5]."Unit Process"."EM - 22X"."FIT22X-1".Address := 276;

END_DATA_BLOCK

